// TwinCAT 3 PLC project AutomatischeDeur
// ProgramVersion: 3.1.4024.0
// libraries:
//   Tc2_Standard, * (Beckhoff Automation GmbH)
//   Tc2_System, * (Beckhoff Automation GmbH)
//   Tc3_Module, * (Beckhoff Automation GmbH)
// project tree:
//   / PlcTask.TcTTO
//   POUs/ MAIN.TcPOU
// (motion and I/O tree: see PLC project trappenhuis_extraverlenging)
// real-time tasks:
//   TASK PlcTask: cycle T#10ms, priority 20, ADS port 350
//   TASK PlcTask1: cycle T#10ms, priority 21, ADS port 351
//   TASK PlcTask2: cycle T#10ms, priority 22, ADS port 352
//   TASK PlcTask3: cycle T#10ms, priority 23, ADS port 353
//   TASK PlcTask4: cycle T#10ms, priority 24, ADS port 354
//   TASK PlcTask5: cycle T#10ms, priority 25, ADS port 355
//   TASK PlcTask6: cycle T#10ms, priority 26, ADS port 356
//   TASK PlcTask7: cycle T#10ms, priority 27, ADS port 357
//   TASK PlcTask8: cycle T#10ms, priority 28, ADS port 358
//   TASK PlcTask9: cycle T#10ms, priority 29, ADS port 359
//   TASK PlcTask10: cycle T#10ms, priority 30, ADS port 360

CONFIGURATION AutomatischeDeur
    RESOURCE PLC ON TwinCAT3
        TASK PlcTask(INTERVAL := T#10ms, PRIORITY := 25);
        PROGRAM MAIN WITH PlcTask : MAIN;
    END_RESOURCE
END_CONFIGURATION

// ---- POUs/MAIN.TcPOU
PROGRAM MAIN
VAR
    bPhotoCell: BOOL; // Boolean variabele voor de fotocel bij de ingang
    bButton: BOOL; // Boolean variabele voor de drukknop bij de kassa
    bMainSwitch: BOOL; // Boolean variabele voor de hoofdschakelaar in het bureau
    fbDoorTimer: TON; // Timer On function block voor de deur
END_VAR

(*
Automatische deur (1 regel code)

Aan een supermarkt wordt de ingangsdeur geopend en gesloten d.m.v. twee pneumatische cilinders. 
Aan de ingang buiten staat een fotocel die de deur zal openen bij een naderende klant.
Ook aan de kassa kan men de deur openen door gebruik te maken van een drukknop.

De deur wordt automatisch gesloten 1 seconde nadat het detectiesignaal is weggevallen.
De automatische werking functioneert enkel als een hoofdschakelaar in het bureau AAN staat.
*)

fbDoorTimer(IN:=(bPhotoCell OR bButton) AND bMainSwitch, PT:=T#1S);

END_PROGRAM
